// TIA Portal V20 export
VAR_GLOBAL   // PLC tag table "TIAC_Inputs_Moteur"
   bStart AT %I0.0 : Bool;
   bStop AT %I0.1 : Bool;
   bFault AT %I0.2 : Bool;
   bRunFeedback AT %I0.3 : Bool;
END_VAR
